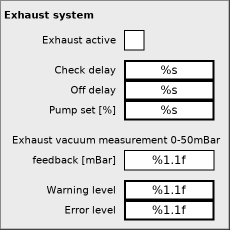
VISUALIZATION _VISU_ExhaustSystemPrint  // 230x230
VAR_IN_OUT
	mInst : FB_ExhaustSystemPrint;
END_VAR
    Rectangle (0,0 230x230)
    Rectangle (1,5 192x20), "Exhaust system"
    Rectangle (29,60 90x20), "Check delay"
    Rectangle (124,60 90x20), "%s", text variable: mInst.tR_VacuumCheckDelay
        OnMouseDown: write the text variable via Edit
    Rectangle (29,80 90x20), "Off delay"
    Rectangle (124,80 90x20), "%s", text variable: mInst.tR_FUOffDelay
        OnMouseDown: write the text variable via Edit
    RoundedRectangle (124,30 20x20), colour toggle: mInst.bO_FUActivate
    Rectangle (19,30 100x20), "Exhaust active"
    Rectangle (9,130 220x20), "Exhaust vacuum measurement 0-50mBar"
    Rectangle (29,150 90x20), "feedback [mBar]"
    Rectangle (124,150 90x20), "%1.1f", text variable: mInst.fL_VacuumAnalogLevelMBar
    Rectangle (29,180 90x20), "Warning level"
    Rectangle (124,180 90x20), "%1.1f", text variable: mInst.fR_VacuumWarningLevelMBar
        OnMouseDown: write the text variable via Edit
    Rectangle (29,200 90x20), "Error level"
    Rectangle (124,200 90x20), "%1.1f", text variable: mInst.fR_VacuumErrorLevelMBar
        OnMouseDown: write the text variable via Edit
    Rectangle (29,100 90x20), "Pump set [%]"
    Rectangle (124,100 90x20), "%s", text variable: mInst.iR_VacuumPumpSetPercent
        OnMouseDown: write the text variable via Edit, min 0, max 100
END_VISUALIZATION

(* stored: Version 1.1.0.1, ProductVersion 3.1.4024.11
   Visu _VISU_ExhaustSystemPrint: Id {5580a83c-e9b0-476c-aa0a-b31bdf4d2059} *)
